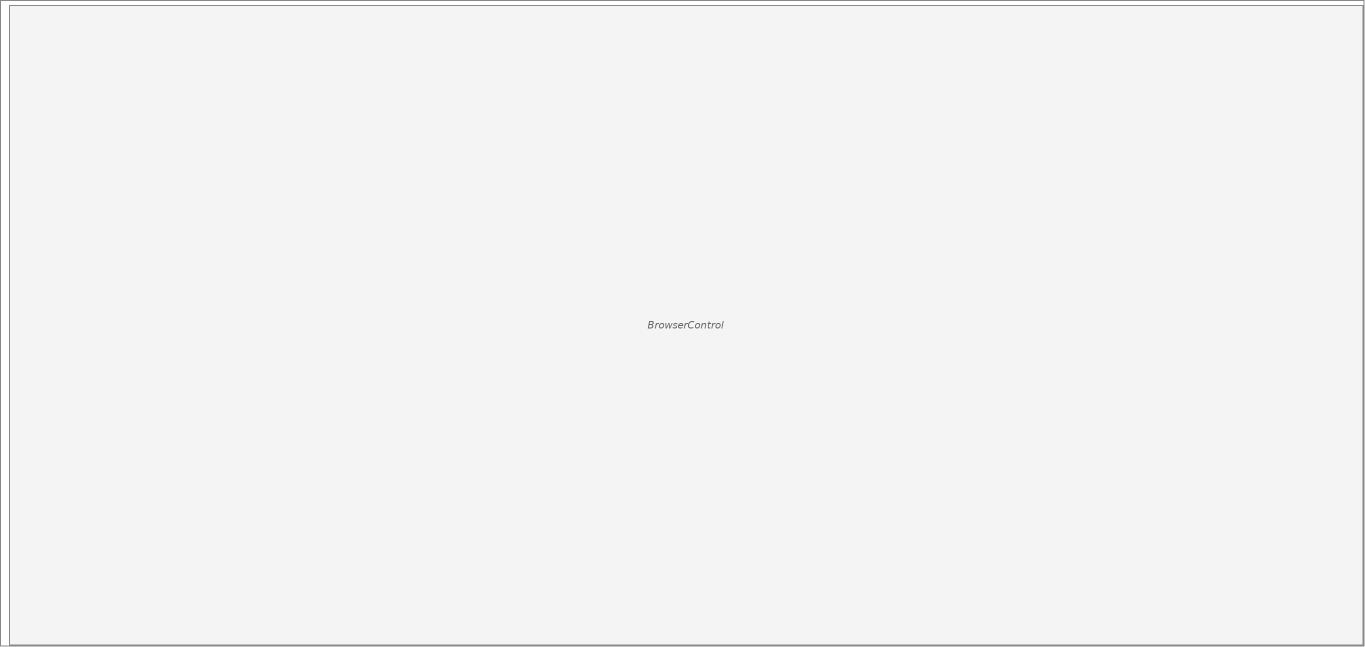
VISUALIZATION ProgramScreen  // 1365x647
    BrowserControl (9,5 1354x640)
        p3734058945: GVL.programURL
END_VISUALIZATION

(* stored: Version 1.1.0.1, ProductVersion 3.1.4022.16
   Visu ProgramScreen: Id {a6649c2f-7194-46ae-81ca-d92d77f74cf0} *)
